// TIA Portal V17 export
// export: Created 2024-09-02T12:50:26.9327523Z, ExportSetting WithDefaults, DisplayName Totally Integrated Automation Portal, DisplayVersion V17, DisplayName TIA Portal Openness, DisplayVersion V17, DisplayName TIA Portal Version Control Interface, DisplayVersion V17, DisplayName STEP 7 Professional, DisplayVersion V17, DisplayName STEP 7 Safety, DisplayVersion V17, DisplayName WinCC Professional, DisplayVersion V17
TYPE "ef_MGB"
// stored: IsFailsafeCompliant true
   STRUCT
      NotHalt : Bool;   // Profisafe - Not-Halt / Profisafe - Emergency stop
      "res5.1" : Bool;   // Profisafe - Reserve
      Türstellung : Bool;   // Profisafe - (T) Türstellung / Profisafe - (T) Door position
      Riegelstellung : Bool;   // Profisafe - (R) Riegelstellung / Profisafe - (R) Blocking position
      Zuhaltung : Bool;   // Profisafe - (Z) Zuhaltung / Profisafe - (Z) guard Blocking
      "res5.5" : Bool;   // Profisafe - Reserve
      "res5.6" : Bool;   // Profisafe - Reserve
      "res5.7" : Bool;   // Profisafe - Reserve
      Sk : Bool;   // Profisafe - SK (T&R)
      Uk : Bool;   // Profisafe - UK (T&R&Z)
      "res6.2" : Bool;   // Profisafe - Reserve
      "res6.3" : Bool;   // Profisafe - Reserve
      "res6.4" : Bool;   // Profisafe - Reserve
      "res6.5" : Bool;   // Profisafe - Reserve
      "res6.6" : Bool;   // Profisafe - Reserve
      "res6.7" : Bool;   // Profisafe - Reserve
      "res7.0" : Bool;   // Profisafe - Reserve
      "res7.1" : Bool;   // Profisafe - Reserve
      "res7.2" : Bool;   // Profisafe - Reserve
      "res7.3" : Bool;   // Profisafe - Reserve
      "res7.4" : Bool;   // Profisafe - Reserve
      "res7.5" : Bool;   // Profisafe - Reserve
      "res7.6" : Bool;   // Profisafe - Reserve
      "res7.7" : Bool;   // Profisafe - Reserve
      "res8.0" : Bool;   // Profisafe - Reserve
      "res8.1" : Bool;   // Profisafe - Reserve
      "res8.2" : Bool;   // Profisafe - Reserve
      "res8.3" : Bool;   // Profisafe - Reserve
      "res8.4" : Bool;   // Profisafe - Reserve
      "res8.5" : Bool;   // Profisafe - Reserve
      "res8.6" : Bool;   // Profisafe - Reserve
      "res8.7" : Bool;   // Profisafe - Reserve
      "res9.0" : Bool;   // Profisafe - Reserve
      "res9.1" : Bool;   // Profisafe - Reserve
      "res9.2" : Bool;   // Profisafe - Reserve
      "res9.3" : Bool;   // Profisafe - Reserve
      "res9.4" : Bool;   // Profisafe - Reserve
      "res9.5" : Bool;   // Profisafe - Reserve
      "res9.6" : Bool;   // Profisafe - Reserve
      "res9.7" : Bool;   // Profisafe - Reserve
      "res10.0" : Bool;   // Profisafe - Reserve
      "res10.1" : Bool;   // Profisafe - Reserve
      "res10.2" : Bool;   // Profisafe - Reserve
      "res10.3" : Bool;   // Profisafe - Reserve
      "res10.4" : Bool;   // Profisafe - Reserve
      "res10.5" : Bool;   // Profisafe - Reserve
      "res10.6" : Bool;   // Profisafe - Reserve
      "res10.7" : Bool;   // Profisafe - Reserve
   END_STRUCT;
END_TYPE
